// TIA Portal V20 export
TYPE "UDT_Service_StepRawDataMedium"
   STRUCT
      "step" : Array[0..99] of "UDT_Service_StepSmall";
      parameterDefinition : Array[0..31] of "UDT_Service_ParameterDefinition";
   END_STRUCT;
END_TYPE
